// TIA Portal project "Lift_2026" (V15.1)

(* hardware
DEVICE "S71500/ET200MP station_1"  S7-1500 station
   slot 0: "Rail_0"  Rack  6ES7 590-1***0-0AA0
   slot 1: "PLC_1"  CPU 1513-1 PN  6ES7 513-1AL02-0AB0  V2.6
      slot 3: "CPU display_1"  6ES7591-1AA00-0AA0
DEVICE "HMI_1"  KTP900 Basic PN
   slot 0: "HMI_1"  KTP900 Basic PN  6AV2 123-2JB03-0AX0  15.1.0.0
   slot 1: "HMI_RT_1"  KTP900 Basic PN  6AV2 123-2JB03-0AX0  15.1.0.0
   slot 5: "HMI_1.IE_CP_1"  PROFINET Interface  15.0.1.0
      slot 1: "PROFINET Interface_1"  PROFINET Interface
         slot 1: "Port_1"  Port
*)

// ===== PLC "PLC_1"  CPU 1513-1 PN =====

DATA_BLOCK "Alarme"   // DB1
{ S7_Optimized_Access := 'TRUE' }
VERSION : 0.1
   VAR
      alarme_gather : Word;
      alarme_vect : Array[0..15] of Bool;
   END_VAR
BEGIN
END_DATA_BLOCK

DATA_BLOCK "Avarii"   // DB2
{ S7_Optimized_Access := 'TRUE' }
VERSION : 0.1
   VAR
      esd : Bool;
      btn_esd : Bool;
      reset_esd : Bool;
      avarie_generala : Bool;
      reset_avarie_generala : Bool;
      avarie_usa : Bool;
      avarie_lumina : Bool;
      avarie_motor : Bool;
      avarie_greutate : Bool;
   END_VAR
BEGIN
END_DATA_BLOCK

DATA_BLOCK "Usa_DB"   // DB3
{ S7_Optimized_Access := 'TRUE' }
VERSION : 0.1
   VAR
      permisiune_plecare : Bool;
      usa_deschisa : Bool;
   END_VAR
BEGIN
END_DATA_BLOCK

DATA_BLOCK "Bec_DB"   // DB4
{ S7_Optimized_Access := 'TRUE' }
VERSION : 0.1
   VAR
      permisiune_pornire : Bool;
      led_aprins : Bool;
   END_VAR
BEGIN
END_DATA_BLOCK

DATA_BLOCK "Motor_DB"   // DB5
{ S7_Optimized_Access := 'TRUE' }
VERSION : 0.1
   VAR
      pornire_stea : Bool;
      pornire_triunghi : Bool;
      motor_pornit : Bool;
      directie_sus : Bool;
      directie_jos : Bool;
      permisiune_plecare : Bool;
   END_VAR
BEGIN
END_DATA_BLOCK

DATA_BLOCK "Simulare_DB"   // DB6
{ S7_Optimized_Access := 'TRUE' }
VERSION : 0.1
   VAR
      directie : USInt;
   END_VAR
BEGIN
END_DATA_BLOCK

DATA_BLOCK "Senzor_greutate_DB"   // DB7
{ S7_Optimized_Access := 'TRUE' }
VERSION : 0.1
   VAR
      permisiune_plecare : Bool;
      greutate_maxima : Real;
      greutate_curenta : Real;
      greutate_depasita : Bool;
   END_VAR
BEGIN
END_DATA_BLOCK

// folder: System blocks/Program resources

DATA_BLOCK "timer_reset_esd"   // DB8
{ S7_Optimized_Access := 'TRUE' }
AUTHOR : Simatic
FAMILY : IEC
NAME : IEC_TMR
VERSION : 1.0
// stored: InstanceOfName IEC_TIMER
"IEC_TIMER"
BEGIN
END_DATA_BLOCK

DATA_BLOCK "timer_reset_avarie_generala"   // DB9
{ S7_Optimized_Access := 'TRUE' }
AUTHOR : Simatic
FAMILY : IEC
NAME : IEC_TMR
VERSION : 1.0
// stored: InstanceOfName IEC_TIMER
"IEC_TIMER"
BEGIN
END_DATA_BLOCK

// folder: (top level)

FUNCTION_BLOCK "Usa"   // FB1, LAD
{ S7_Optimized_Access := 'TRUE' }
VERSION : 0.1
   VAR_INPUT
      permisiune_plecare : Bool;
   END_VAR
   VAR_OUTPUT
      usa_deschisa : Bool;
   END_VAR
BEGIN

REGION Network 1
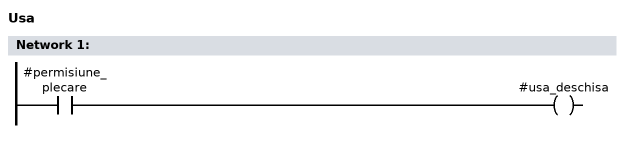
   RUNG wire#powerrail
      Contact( #permisiune_plecare )
      Coil( #usa_deschisa )
   END_RUNG
   // the same network as SCL:
   #usa_deschisa := #permisiune_plecare;
END_REGION
END_FUNCTION_BLOCK

FUNCTION_BLOCK "Bec"   // FB2, LAD
{ S7_Optimized_Access := 'TRUE' }
VERSION : 0.1
   VAR_INPUT
      permisiune_pornire : Bool;
   END_VAR
   VAR_OUTPUT
      bec_aprins : Bool;
   END_VAR
BEGIN

REGION Network 1
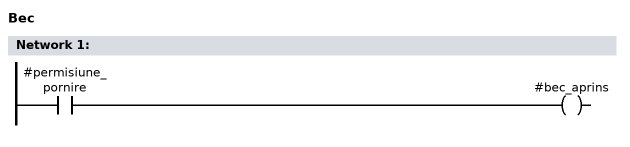
   RUNG wire#powerrail
      Contact( #permisiune_pornire )
      Coil( #bec_aprins )
   END_RUNG
   // the same network as SCL:
   #bec_aprins := #permisiune_pornire;
END_REGION
END_FUNCTION_BLOCK

FUNCTION_BLOCK "Motor"   // FB3, LAD
{ S7_Optimized_Access := 'TRUE' }
VERSION : 0.1
   VAR_INPUT
      directie : USInt;
   END_VAR
   VAR_OUTPUT
      pornire_stea : Bool;
      pornire_triunghi : Bool;
      motor_pornit : Bool;
      directie_sus : Bool;
      directie_jos : Bool;
   END_VAR
   VAR_IN_OUT
      permisiune_plecare : Bool;
   END_VAR
   VAR
      timer_stea : TON_TIME;
      plecare_sus : Bool;
      plecare_jos : Bool;
   END_VAR
BEGIN

REGION Network 1: Selecteaza directia
   // simulata cu valori algebrice, insa in mod normal ar fi un contact pentru directie, depinzand cum se conecteaza, selecteaza directia, insa pentru simplitate am optat la asta)
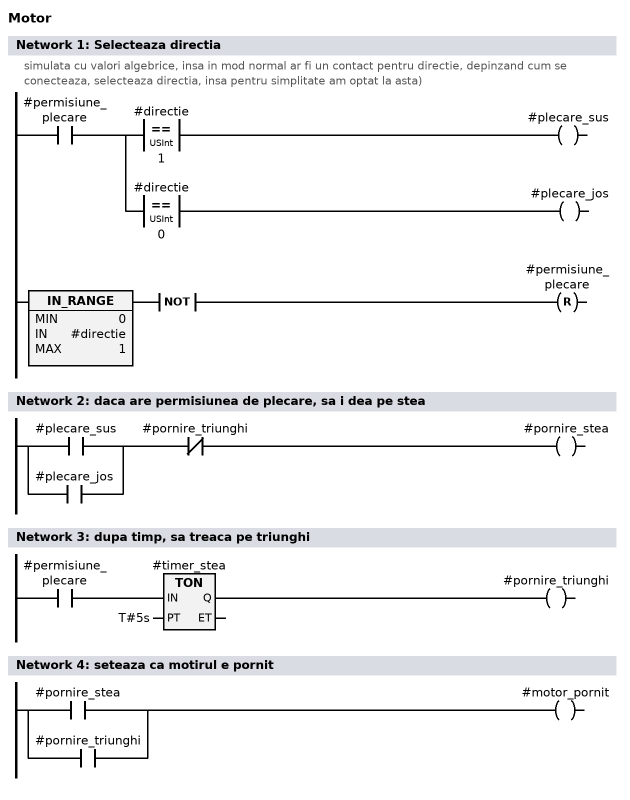
   RUNG wire#powerrail
      Contact( #permisiune_plecare )
      wire#w1
      { S7_Templates := "SrcType := USInt" } EQ_Contact(in1 := #directie, in2 := 1)
      Coil( #plecare_sus )
   END_RUNG
   RUNG wire#w1
      { S7_Templates := "SrcType := USInt" } EQ_Contact(in1 := #directie, in2 := 0)
      Coil( #plecare_jos )
   END_RUNG
   RUNG wire#powerrail
      { S7_Templates := "SrcType := USInt" } InRange(min := 0, in := #directie, max := 1)
      Not()
      R_Coil( #permisiune_plecare )
   END_RUNG
   // the same network as SCL:
   #plecare_sus := #permisiune_plecare AND (#directie = 1);
   #plecare_jos := #permisiune_plecare AND (#directie = 0);
   IF NOT ((0 <= #directie) AND (#directie <= 1)) THEN #permisiune_plecare := FALSE; END_IF;
END_REGION

REGION Network 2: daca are permisiunea de plecare, sa i dea pe stea
   RUNG wire#powerrail
      Contact( #plecare_sus )
      wire#w1
      I_Contact( #pornire_triunghi )
      Coil( #pornire_stea )
   END_RUNG
   RUNG wire#powerrail
      Contact( #plecare_jos )
   END_RUNG wire#w1
   // the same network as SCL:
   #pornire_stea := (#plecare_sus OR #plecare_jos) AND NOT #pornire_triunghi;
END_REGION

REGION Network 3: dupa timp, sa treaca pe triunghi
   #timer_stea(IN := #permisiune_plecare, PT := T#5s);   // TON
   #pornire_triunghi := #timer_stea.Q;
END_REGION

REGION Network 4: seteaza ca motirul e pornit
   RUNG wire#powerrail
      Contact( #pornire_stea )
      wire#w1
      Coil( #motor_pornit )
   END_RUNG
   RUNG wire#powerrail
      Contact( #pornire_triunghi )
   END_RUNG wire#w1
   // the same network as SCL:
   #motor_pornit := #pornire_stea OR #pornire_triunghi;
END_REGION
END_FUNCTION_BLOCK

FUNCTION_BLOCK "Simulare"   // FB4, LAD
{ S7_Optimized_Access := 'TRUE' }
VERSION : 0.1
BEGIN
END_FUNCTION_BLOCK

FUNCTION_BLOCK "Senzor_greutate"   // FB5, LAD
{ S7_Optimized_Access := 'TRUE' }
VERSION : 0.1
   VAR_INPUT
      permisiune_plecare : Bool;
      greutate_maxima : Real;
   END_VAR
   VAR_OUTPUT
      greutate_curenta : Real;
      greutate_depasita : Bool;
   END_VAR
   VAR
      pornit : Bool;
   END_VAR
BEGIN

REGION Network 1: daca are permisiune de plecare,
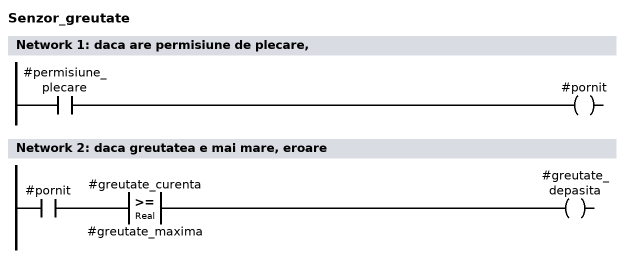
   RUNG wire#powerrail
      Contact( #permisiune_plecare )
      Coil( #pornit )
   END_RUNG
   // the same network as SCL:
   #pornit := #permisiune_plecare;
END_REGION

REGION Network 2: daca greutatea e mai mare, eroare
   RUNG wire#powerrail
      Contact( #pornit )
      { S7_Templates := "SrcType := Real" } GE_Contact(in1 := #greutate_curenta, in2 := #greutate_maxima)
      Coil( #greutate_depasita )
   END_RUNG
   // the same network as SCL:
   #greutate_depasita := #pornit AND (#greutate_curenta >= #greutate_maxima);
END_REGION
END_FUNCTION_BLOCK

ORGANIZATION_BLOCK "Main"   // OB1, LAD, ProgramCycle
TITLE = "Main Program Sweep (Cycle)"
{ S7_Optimized_Access := 'TRUE' }
VERSION : 0.1
   VAR_INPUT
      Initial_Call : Bool;   // Initial call of this OB
      Remanence : Bool;   // =True, if remanent data are available
   END_VAR
BEGIN

REGION Network 1: Alarme gather
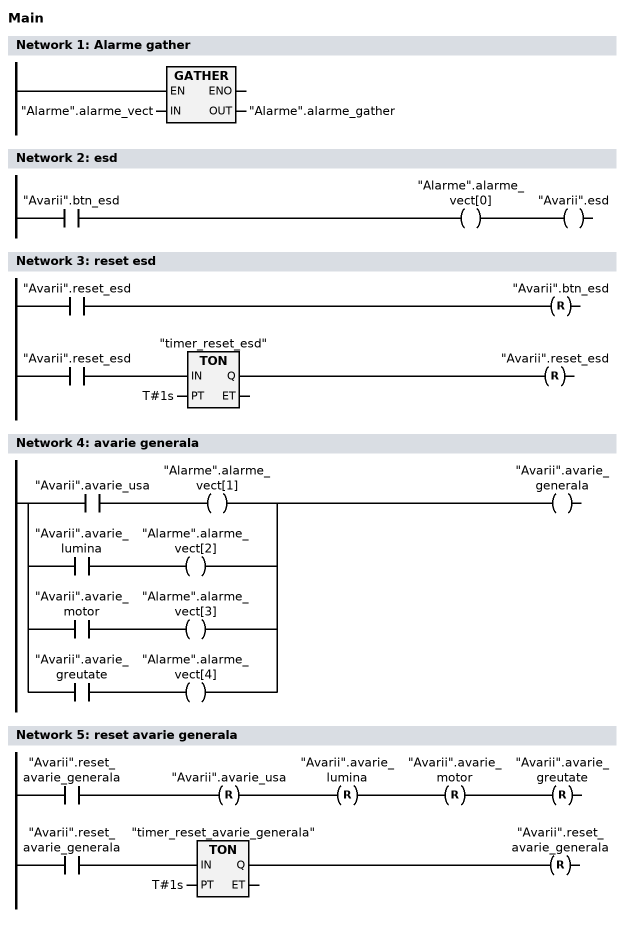
   GATHER(IN := "Alarme".alarme_vect, OUT => "Alarme".alarme_gather);
END_REGION

REGION Network 2: esd
   RUNG wire#powerrail
      Contact( "Avarii".btn_esd )
      Coil( "Alarme".alarme_vect[0] )
      Coil( "Avarii".esd )
   END_RUNG
   // the same network as SCL:
   "Alarme".alarme_vect[0] := "Avarii".btn_esd;
   "Avarii".esd := "Avarii".btn_esd;
END_REGION

REGION Network 3: reset esd
   IF "Avarii".reset_esd THEN "Avarii".btn_esd := FALSE; END_IF;
   "timer_reset_esd".TON(IN := "Avarii".reset_esd, PT := T#1s);
   IF "timer_reset_esd".Q THEN "Avarii".reset_esd := FALSE; END_IF;
END_REGION

REGION Network 4: avarie generala
   RUNG wire#powerrail
      Contact( "Avarii".avarie_usa )
      Coil( "Alarme".alarme_vect[1] )
      wire#w1
      Coil( "Avarii".avarie_generala )
   END_RUNG
   RUNG wire#powerrail
      Contact( "Avarii".avarie_lumina )
      Coil( "Alarme".alarme_vect[2] )
   END_RUNG wire#w1
   RUNG wire#powerrail
      Contact( "Avarii".avarie_motor )
      Coil( "Alarme".alarme_vect[3] )
   END_RUNG wire#w1
   RUNG wire#powerrail
      Contact( "Avarii".avarie_greutate )
      Coil( "Alarme".alarme_vect[4] )
   END_RUNG wire#w1
   // the same network as SCL:
   "Alarme".alarme_vect[1] := "Avarii".avarie_usa;
   "Alarme".alarme_vect[2] := "Avarii".avarie_lumina;
   "Alarme".alarme_vect[3] := "Avarii".avarie_motor;
   "Alarme".alarme_vect[4] := "Avarii".avarie_greutate;
   "Avarii".avarie_generala := "Avarii".avarie_usa OR "Avarii".avarie_lumina OR "Avarii".avarie_motor OR "Avarii".avarie_greutate;
END_REGION

REGION Network 5: reset avarie generala
   IF "Avarii".reset_avarie_generala THEN
       "Avarii".avarie_usa := FALSE;
       "Avarii".avarie_lumina := FALSE;
       "Avarii".avarie_motor := FALSE;
       "Avarii".avarie_greutate := FALSE;
   END_IF;
   "timer_reset_avarie_generala".TON(IN := "Avarii".reset_avarie_generala, PT := T#1s);
   IF "timer_reset_avarie_generala".Q THEN "Avarii".reset_avarie_generala := FALSE; END_IF;
END_REGION
END_ORGANIZATION_BLOCK

(* ===== HMI "HMI_RT_1" =====
system functions are stored by id; their names below are inferred from use
connection "HMI_Connection_1": ETHERNET, SMART_S7_1500_OMS

HMI tags "Default tag table"
   "Alarme_alarme_gather" : Word = PLC Alarme.alarme_gather, 1 s

discrete alarms
   1: 'ESD', class Errors, trigger "Alarme_alarme_gather" bit 0
   2: 'Avarie la usa', class Errors, trigger "Alarme_alarme_gather" bit 1
   3: 'Avarie la bec', class Errors, trigger "Alarme_alarme_gather" bit 2
   4: 'Avarie la motor', class Errors, trigger "Alarme_alarme_gather" bit 3
   5: 'Avarie la senzorul de greutate', class Errors, trigger "Alarme_alarme_gather" bit 4
   6: '', class Errors, trigger "Alarme_alarme_gather" bit 5

Template "Template_1" 800x480
   Button "Exit" at 722,440 size 55x39; TextOff 'Exit'; PictureOff "ExitRuntime_KTP900_Basic_PN_TR"; PictureOn "ExitRuntime_KTP900_Basic_PN_TR"
      on Release: StopRuntime(0)
   Button "Template_Button" at 622,440 size 55x39; TextOff 'Text'
   Button "Template_Button_1" at 522,440 size 55x39; TextOff 'Text'
   Button "Template_Button_2" at 422,440 size 55x39; TextOff 'Text'
   Button "Template_Button_3" at 322,440 size 55x39; TextOff 'Text'
   Button "Template_Button_4" at 222,440 size 55x39; TextOff 'Text'
   Button "Template_Button_5" at 122,440 size 55x39; TextOff 'Text'
   Button "Start screen" at 22,440 size 55x39; TextOff 'Start screen'; PictureOff "NavigateHome_KTP900_Basic_PN_TR"; PictureOn "NavigateHome_KTP900_Basic_PN_TR"
      on Release: ActivateScreen("Main", 0)
*)